FUNCTION_BLOCK FB_SMSDatasetFifo_Read
VAR_INPUT
    bOverwrite : BOOL;
    In         : ST_SMSDataSetEntry_Read;
END_VAR
VAR_OUTPUT
    bOk        : BOOL;
    nCount     : UDINT;
    nLoad      : UDINT;
    Out        : ST_SMSDataSetEntry_Read;
END_VAR
VAR
    arrBuffer  : ARRAY[0..Max_buffer_size_G] OF BYTE; (* Buffer memory used by FB_MemRingBuffer function block *)
    fbBuffer   : FB_MemRingBuffer;
END_VAR

ACTION A_Add:
fbBuffer.A_AddTail(pWrite := ADR(in),
						   cbWrite:=SIZEOF(in),
						   pBuffer:=ADR(arrBuffer),
						   cbBuffer:=SIZEOF(arrBuffer),
						   bOK=>bOK,
						   nCount =>nCount);
IF NOT bOK THEN 
	IF bOverwrite THEN
		fbBuffer.A_RemoveHead();(*remove one oldest entry*)
		fbBuffer.A_AddTail(bOK => bOk,nCount => nCount);
	END_IF
END_IF

nload := (fbbuffer.cbSize * 100)/(Max_buffer_size_G);
END_ACTION

ACTION A_Get:
fbBuffer.A_GetHead(pWrite := ADR(out),
						   cbWrite:=SIZEOF(out),
						   pBuffer:=ADR(arrBuffer),
						   cbBuffer:=SIZEOF(arrBuffer),
						   bOK=>bOK,
						   nCount =>nCount);
nload := (fbbuffer.cbSize * 100)/(Max_buffer_size_G);
END_ACTION

ACTION A_Remove:
fbBuffer.A_RemoveHead(pRead:=ADR(out),
						cbRead:=SIZEOF(out),
						pBuffer:=ADR(arrBuffer),
						cbBuffer:=SIZEOF(arrBuffer),
						bOK=>bOK,
						nCount =>nCount);
nload := (fbbuffer.cbSize * 100)/(Max_buffer_size_G);
END_ACTION

ACTION A_Reset:
MEMSET(ADR(arrBuffer),0,SIZEOF(arrBuffer)); (*reset internal buffer*)
fbBuffer.A_Reset(bOK=>bOK,nCount=>ncount);
nload := (fbbuffer.cbSize * 100)/(Max_buffer_size_G);
END_ACTION

END_FUNCTION_BLOCK

(* stored: Version 1.1.0.1, ProductVersion 3.1.4024.6
   POU FB_SMSDatasetFifo_Read: Id {93b7e475-4d36-4275-9cff-239a481a2e13}, SpecialFunc None
   Action A_Add: Id {94363380-9844-4b6e-b189-25074ac4fbb5}
   Action A_Get: Id {b1fda7ed-843f-4350-a563-2fea4b7f2166}
   Action A_Remove: Id {c9e8751f-6d67-406d-9dad-f3238791af41}
   Action A_Reset: Id {27452247-78c6-4489-b324-a3887ba2f787} *)
